// TIA Portal V20 export
// export: Created 2025-12-01T14:57:24.2646503Z, ExportSetting None, DisplayName Totally Integrated Automation Portal, DisplayVersion V20 Update 3, DisplayName TIA Portal Openness, DisplayVersion V20 Update 3, DisplayName TIA Portal Version Control Interface, DisplayVersion V20 Update 3, DisplayName STEP 7 Professional, DisplayVersion V20 Update 3, DisplayName STEP 7 Safety, DisplayVersion V20 Update 2, DisplayName WinCC Basic/Comfort/Advanced, DisplayVersion V20 Update 3, DisplayName WinCC Professional, DisplayVersion V20 Update 3, DisplayName WinCC Unified, DisplayVersion V20 Update 3
FUNCTION "FC962_ScadaZona" : Void   // FC962, STL
{ S7_Optimized_Access := 'FALSE' }
AUTHOR : SCADA
NAME : 20161001
VERSION : 1.0
// stored: AutoNumber false
   VAR_INPUT
      NumZona : UInt;
      P_Marcha : Bool;
      P_Paro : Bool;
      P_Rearme : Bool;
      P_TestLuces : Bool;
      P_Auto : Bool;
      P_OffLine : Bool;
      P_Main : Bool;
      H_Verde : Bool;
      H_Roja : Bool;
      H_Naranja : Bool;
   END_VAR
   VAR_TEMP
      ValorReturn : Int;
      Zona : UInt;
   END_VAR
BEGIN

NETWORK
TITLE = Inicializar
////////////////////////////////////////////////////////////////////////////////
////////////////////////////////////////////////////////////////////////////////
////////////////////////////////////////////////////////////////////////////////
// --- Tareas Iniciales
      L     #NumZona;  // Numero de Zona a tratar
      T     #Zona;



NETWORK
TITLE = Transferencia del Estado de la Zona
////////////////////////////////////////////////////////////////////////////////
////////////////////////////////////////////////////////////////////////////////
////////////////////////////////////////////////////////////////////////////////
// --- Transferencia: Estado de la Zona, Codigo de Error
      CALL  BLKMOV
      ( SRCBLK  := "DB901_Estado_Zonas".EstadoZona[#Zona].Estado,
        RET_VAL := #ValorReturn,
        DSTBLK  := "DB013_ScadaZona".Zona[#Zona].Estado
      );

      CALL  MOVE
      ( IN  := "DB901_Estado_Zonas".EstadoZona[#Zona].CodigoError,
        OUT := "DB013_ScadaZona".Zona[#Zona].CodigoError
      );



NETWORK
TITLE = Transferencia de Entradas
////////////////////////////////////////////////////////////////////////////////
////////////////////////////////////////////////////////////////////////////////
////////////////////////////////////////////////////////////////////////////////
// --- Transferencia de las Entrada
      SET;
      A     #P_Marcha;  // - Pulsador de Marcha
      =     "DB013_ScadaZona".Zona[#Zona].Entradas.Marcha;

      SET;
      A     #P_Paro;  // - Pulsador de Paro
      =     "DB013_ScadaZona".Zona[#Zona].Entradas.Paro;

      SET;
      A     #P_Rearme;  // - Pulsador de Rearme
      =     "DB013_ScadaZona".Zona[#Zona].Entradas.Rearme;

      SET;
      A     #P_Auto;  // - Selector de Auto
      =     "DB013_ScadaZona".Zona[#Zona].Entradas.Auto;

      SET;
      A     #P_TestLuces;  // - Pulsador de TestLuces
      =     "DB013_ScadaZona".Zona[#Zona].Entradas.TestLuces;

      SET;
      A     #P_OffLine;  // - Selector de Off Line
      =     "DB013_ScadaZona".Zona[#Zona].Entradas.Off_Line;

      SET;
      A     #P_Main;  // - Selector de Maintenimineto
      =     "DB013_ScadaZona".Zona[#Zona].Entradas.Maintenimiento;



NETWORK
TITLE = Transferencia de Salidas
////////////////////////////////////////////////////////////////////////////////
////////////////////////////////////////////////////////////////////////////////
////////////////////////////////////////////////////////////////////////////////
// ---  Transferencia de Salidas

      SET;
      A     #H_Verde;  // - Baliza Verde
      =     "DB013_ScadaZona".Zona[#Zona].Salidas.H_Verde;

      SET;
      A     #H_Roja;  // - Baliza Roja
      =     "DB013_ScadaZona".Zona[#Zona].Salidas.H_Roja;

      SET;
      A     #H_Naranja;  // - Baliza Naranja
      =     "DB013_ScadaZona".Zona[#Zona].Salidas.H_Naranja;



NETWORK
TITLE = Transferencia de Datos de Scada
////////////////////////////////////////////////////////////////////////////////
////////////////////////////////////////////////////////////////////////////////
////////////////////////////////////////////////////////////////////////////////
// --- Transferencia de la Primera Parte


      SET;  // - Aviso de Emergencia Grave
      A     "DB901_Estado_Zonas".EstadoZona[#Zona].Pulsador.EmergenciaGrave;
      =     "DB013_ScadaZona".Zona[#Zona].DatosScada.EmergenciaGrave;

      SET;  // - Aviso de Energencia Leve
      A     "DB901_Estado_Zonas".EstadoZona[#Zona].Pulsador.EmergenciaLeve;
      =     "DB013_ScadaZona".Zona[#Zona].DatosScada.EmergenciaLeve;

      SET;  // - Aviso de Error Grave
      A     "DB901_Estado_Zonas".EstadoZona[#Zona].Pulsador.ErrorGrave;
      =     "DB013_ScadaZona".Zona[#Zona].DatosScada.ErrorGrave;

      SET;  // - Aviso de Error Leve
      A     "DB901_Estado_Zonas".EstadoZona[#Zona].Pulsador.ErrorLeve;
      =     "DB013_ScadaZona".Zona[#Zona].DatosScada.ErrorLeve;

      SET;  // - Fin Reset de la Zona
      A     "DB901_Estado_Zonas".EstadoZona[#Zona].Pulsador.FinReset;
      =     "DB013_ScadaZona".Zona[#Zona].DatosScada.FinReset;

      SET;  // - Memoria Pulsador Marcha
      A     "DB901_Estado_Zonas".EstadoZona[#Zona].Pulsador.MemoriaPulsadorMarcha;
      =     "DB013_ScadaZona".Zona[#Zona].DatosScada.Memo_P_Marcha;

      SET;  // - Memoria Pulsador Paro
      A     "DB901_Estado_Zonas".EstadoZona[#Zona].Pulsador.MemoriaPulsadorParo;
      =     "DB013_ScadaZona".Zona[#Zona].DatosScada.Memo_P_Paro;


////////////////////////////////////////////////////////////////////////////////
////////////////////////////////////////////////////////////////////////////////
////////////////////////////////////////////////////////////////////////////////
// --- Transferencia de la Segunda Parte

      SET;  // - Alguna mesa de la zona en Paro
      A     "DB901_Estado_Zonas".EstadoZona[#Zona].VariablesInternas.MesasParo;
      =     "DB013_ScadaZona".Zona[#Zona].DatosScada.MesasParo;

      SET;  // - Alguna mesa de la zona en Manual
      A     "DB901_Estado_Zonas".EstadoZona[#Zona].VariablesInternas.MesasManual;
      =     "DB013_ScadaZona".Zona[#Zona].DatosScada.MesasManual;

      SET;  // - Alguna mesa de la zona en Paro Blando
      A     "DB901_Estado_Zonas".EstadoZona[#Zona].VariablesInternas.MesasBlando;
      =     "DB013_ScadaZona".Zona[#Zona].DatosScada.MesasParoBlando;

      SET;  // - Alguna mesa de la zona en Error
      A     "DB901_Estado_Zonas".EstadoZona[#Zona].VariablesInternas.MesasError;
      =     "DB013_ScadaZona".Zona[#Zona].DatosScada.MesasError;

      SET;  // - Todas las mesas de la zona en Paro
      A     "DB901_Estado_Zonas".EstadoZona[#Zona].VariablesInternas.MesasTodasParo;
      =     "DB013_ScadaZona".Zona[#Zona].DatosScada.MesasTodasEnParo;

      SET;  // - Todas las mesas de la zona en Manual
      A     "DB901_Estado_Zonas".EstadoZona[#Zona].VariablesInternas.MesasTodasManual;
      =     "DB013_ScadaZona".Zona[#Zona].DatosScada.MesasTodasEnManual;



NETWORK
TITLE = Transferencia de Bits de Emergencias
////////////////////////////////////////////////////////////////////////////////
////////////////////////////////////////////////////////////////////////////////
////////////////////////////////////////////////////////////////////////////////

      CALL  BLKMOV
      ( SRCBLK  := "DB860_Bits_ErroresArmarios".Armarios[#Zona].Emergencias,
        RET_VAL := #ValorReturn,
        DSTBLK  := "DB013_ScadaZona".Zona[#Zona].EmergenciasGraves
      );  // ---  Emergencias Graves



NETWORK
TITLE = Transferencia de Bits de Errores
////////////////////////////////////////////////////////////////////////////////
////////////////////////////////////////////////////////////////////////////////
////////////////////////////////////////////////////////////////////////////////

      CALL  BLKMOV
      ( SRCBLK  := "DB860_Bits_ErroresArmarios".Armarios[#Zona].ErroresGraves,
        RET_VAL := #ValorReturn,
        DSTBLK  := "DB013_ScadaZona".Zona[#Zona].ErroresGraves
      );  // ---  Errores Graves

      CALL  BLKMOV
      ( SRCBLK  := "DB860_Bits_ErroresArmarios".Armarios[#Zona].ErroresLeves,
        RET_VAL := #ValorReturn,
        DSTBLK  := "DB013_ScadaZona".Zona[#Zona].ErroresLeves
      );  // ---  Errores Leves



NETWORK
TITLE = Final de la Funcion
////////////////////////////////////////////////////////////////////////////////
////////////////////////////////////////////////////////////////////////////////
////////////////////////////////////////////////////////////////////////////////
// --- Tareas finales


END_FUNCTION
